SUBAPPLICATION Uebung_052 (* DigitalInput_I1-_I4 auf DigitalOutput_Q1-_Q4 *)
  (* Standard: 61499-2 *)
  (* Version 1.0, 2023-10-23, franz *)
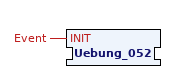
  EVENT_INPUT
    INIT;
  END_EVENT
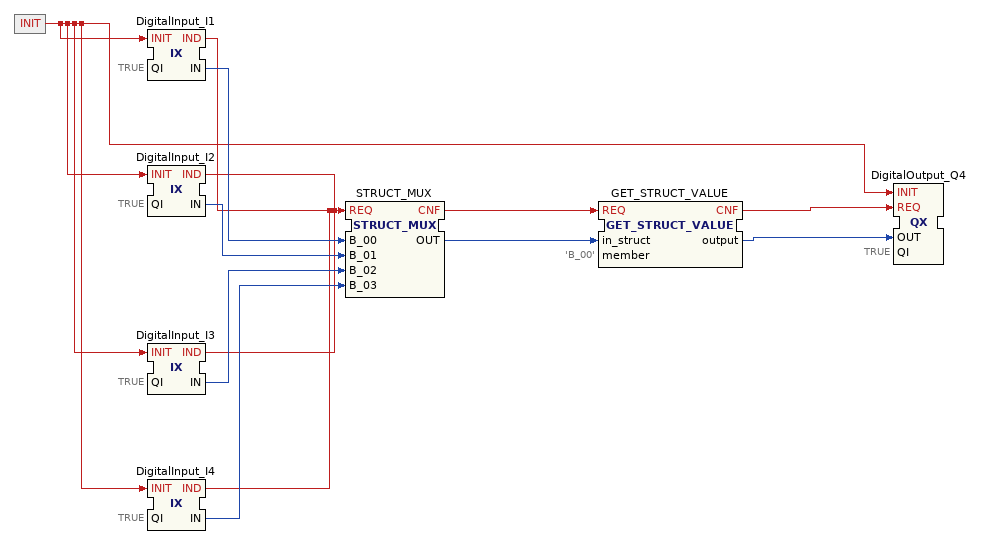
  FBS
    DigitalInput_I1 : IX(QI := TRUE);
    DigitalInput_I2 : IX(QI := TRUE);
    DigitalInput_I3 : IX(QI := TRUE);
    DigitalOutput_Q4 : QX(QI := TRUE);
    DigitalInput_I4 : IX(QI := TRUE);
    GET_STRUCT_VALUE : GET_STRUCT_VALUE(member := 'B_00');
    STRUCT_MUX : STRUCT_MUX(B_00 :=  (* BIT 00 *), B_01 :=  (* BIT 01 *), B_02 :=  (* BIT 02 *), B_03 :=  (* BIT 03 *)); {SET_ATTRIBUTE(StructuredType, ST04B)}
  END_FBS
  EVENT_CONNECTIONS
    INIT TO DigitalInput_I1.INIT;
    INIT TO DigitalInput_I2.INIT;
    INIT TO DigitalInput_I3.INIT;
    INIT TO DigitalInput_I4.INIT;
    INIT TO DigitalOutput_Q4.INIT;
    GET_STRUCT_VALUE.CNF TO DigitalOutput_Q4.REQ;
    DigitalInput_I1.IND TO STRUCT_MUX.REQ;
    DigitalInput_I2.IND TO STRUCT_MUX.REQ;
    DigitalInput_I3.IND TO STRUCT_MUX.REQ;
    DigitalInput_I4.IND TO STRUCT_MUX.REQ;
    STRUCT_MUX.CNF TO GET_STRUCT_VALUE.REQ;
  END_CONNECTIONS
  DATA_CONNECTIONS
    GET_STRUCT_VALUE.output TO DigitalOutput_Q4.OUT;
    DigitalInput_I1.IN TO STRUCT_MUX.B_00;
    DigitalInput_I2.IN TO STRUCT_MUX.B_01;
    DigitalInput_I3.IN TO STRUCT_MUX.B_02;
    DigitalInput_I4.IN TO STRUCT_MUX.B_03;
    STRUCT_MUX.OUT TO GET_STRUCT_VALUE.in_struct;
  END_CONNECTIONS
END_SUBAPPLICATION
